PROGRAM Comp01_Main

Comp01.StateManager ();
Comp01_Sequencer();
Comp01_Devices();

IF Intfc.Upstream_LaneA_Receiver.iHandshake.WaitingToSend THEN
	
END_IF

END_PROGRAM

(* stored: Version 1.1.0.1, ProductVersion 3.1.4022.11
   POU Comp01_Main: Id {baec4577-6414-4931-9ca3-5879091ea58e}, SpecialFunc None *)
